ADAPTER EVENT_HS_UNI_WSTRING (* Handshake family, unidirectional fire-and-forget with WSTRING payload: REQ/REQD only, no reply *)
  (* Standard: 61499-1; Description: Copyright (c) 2026 HR Agrartechnik GmbH This program and the accompanying materials are made available under the terms of the Eclipse Public License 2.0 which is available at https://www.eclipse.org/legal/epl-2.0/ SPDX-License-Identifier: EPL-2.0 *)
  (* Version 1.0, 2026-09-02, Franz Höpfinger, HR Agrartechnik GmbH, Data-carrying variant of EVENT_HS_UNI: adds a WSTRING payload (REQD) to the fire-and-forget REQ, matching the 'name,value' message style (e.g. push,100) documented in HandshakePattern.md *)
  PACKAGE adapter::types::bidirectional::Handshake;
  (* Documentation:
  Data-carrying variant of EVENT_HS_UNI (reduced, unidirectional member of the EVENT_HS family, Handshake design pattern, IEC 61499 primer course, Module 6, Valeriy Vyatkin). Declares a single REQ/REQD event+payload pair, from Plug to Socket - no CNF/CNFD, IND/INDD, or RSP/RSPD at all.
   This is deliberately not a real handshake: the Socket side has no way to acknowledge or refuse the request (or its payload), and the Plug side has no way to know whether the Socket ever received or reacted to it. Use this only for genuine fire-and-forget notifications carrying a payload where that one-way, best-effort semantics is actually acceptable.
   Same Socket/Plug role split as EVENT_HS: Plug (Name>>) keeps the declared direction and fires REQ/REQD; Socket (>>Name) mirrors it and reacts to REQ/REQD.
   See test_AX/Meins/DesingPatterns/HandshakePattern/HandshakePattern.md for the full write-up of the EVENT_HS family, including this and the other three reduced variants (EVENT_HS_UNI, EVENT_HS_ACK, EVENT_HS_ACK_WSTRING).
   The <Service> block below is purely documentation (a service-sequence diagram, per the XSD's minOccurs="0" - optional, not required for the adapter connection to actually forward events; the standard 4diac AE.adp has none either). Added anyway since it does not hurt and makes the single REQ transaction explicit.
  *)
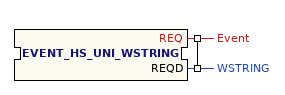
  EVENT_OUTPUT
    REQ WITH REQD; (* Request/notification from Plug to Socket, no reply expected *)
  END_EVENT
  VAR_OUTPUT
    REQD : WSTRING; (* Request payload, accompanies REQ *)
  END_VAR
  SERVICE PLUG/SOCKET
    SEQUENCE notify
      PLUG.REQ(REQD) -> SOCKET.REQ(REQD);
    END_SEQUENCE
  END_SERVICE
END_ADAPTER
